FUNCTION F_ChkSettingLimitN : BOOL
VAR_IN_OUT
	nValue		: INT;
	stSetting 	: ST_Data_Item;
END_VAR
VAR_OUTPUT
	stInfo 		: ST_Text;
END_VAR

F_ChkSettingLimitN := FALSE;

IF (stSetting.eDataType = E_DataType.eDataType_int) AND nValue > stSetting.fValueMax THEN
	stInfo.wsName := "input to high";
	stInfo.wsNameId := "inputtohigh";
	RETURN;
END_IF

IF (stSetting.eDataType = E_DataType.eDataType_int) AND nValue < stSetting.fValueMin THEN
	stInfo.wsName := "input to low";
	stInfo.wsNameId := "inputtolow";
	RETURN;
END_IF

IF (stSetting.eDataType = E_DataType.eDataType_time_ms) AND nValue > stSetting.fValueMax THEN
	stInfo.wsName := "input to high";
	stInfo.wsNameId := "inputtohigh";
	RETURN;
END_IF

IF (stSetting.eDataType = E_DataType.eDataType_time_ms) AND nValue < stSetting.fValueMin THEN
	stInfo.wsName := "input to low";
	stInfo.wsNameId := "inputtolow";
	RETURN;
END_IF

F_ChkSettingLimitN := TRUE;

END_FUNCTION

(* stored: Version 1.1.0.1, ProductVersion 3.1.4024.12
   POU F_ChkSettingLimitN: Id {b19b7468-a75c-495c-b140-b7b52985993e}, SpecialFunc None *)
